FUNCTION_BLOCK Test_TExecutionWhenBusy_Abort_SelectsAborting EXTENDS T_UnitTestbase
VAR
    Execution : T_Execution;
END_VAR

METHOD Init
Execution.FB_init(bInitRetains := FALSE,
                  bInCopyCode  := FALSE);
END_METHOD

{attribute 'analysis' := '-33'} // inhibit unused variable warning
METHOD RunTest
VAR_OUTPUT
    TestCompleted : BOOL;
    TestFailed    : BOOL;
END_VAR
Execution.Start();
Execution.SetBusy();
Execution.Abort();

TestFailed S= NOT AssertTrue(Source    := TestName,
                             Condition := Execution.Aborting,
                             Message   := 'Execution.Aborting not true');

TestCompleted := TRUE;
END_METHOD

END_FUNCTION_BLOCK

(* stored: Version 1.1.0.1, ProductVersion 3.1.4024.12
   POU Test_TExecutionWhenBusy_Abort_SelectsAborting: Id {6aa2306c-ed22-4a07-beed-a9481480c75d}, SpecialFunc None
   Method Init: Id {7d2cb2a3-6dbe-4722-b6b5-d0eb4c0e79db}
   Method RunTest: Id {f1dc014c-f1ac-4f15-8775-88aed48a9767} *)
